FUNCTION_BLOCK SS0 (* Composite FB wrapping other FBs *)
  (* Standard: 61499-2 *)
  (* Version 1.0, 2024-08-30, DEVIASH *)
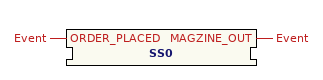
  EVENT_INPUT
    ORDER_PLACED; (* Initialization Request *)
  END_EVENT
  EVENT_OUTPUT
    MAGZINE_OUT; (* Initialization Confirm *)
  END_EVENT
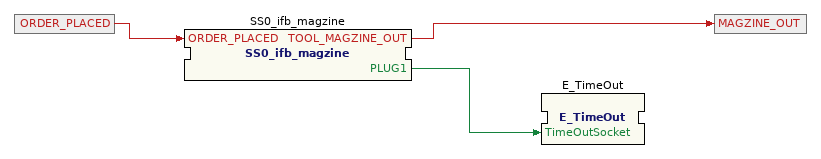
  FBS
    E_TimeOut : E_TimeOut;
    SS0_ifb_magzine : SS0_ifb_magzine;
  END_FBS
  EVENT_CONNECTIONS
    ORDER_PLACED TO SS0_ifb_magzine.ORDER_PLACED;
    SS0_ifb_magzine.TOOL_MAGZINE_OUT TO MAGZINE_OUT;
  END_CONNECTIONS
  ADAPTER_CONNECTIONS
    SS0_ifb_magzine.PLUG1 TO E_TimeOut.TimeOutSocket;
  END_CONNECTIONS
END_FUNCTION_BLOCK
